INTERFACE IReadOnlyListOfBytes EXTENDS IPointerCollection

METHOD Find : BOOL
VAR_INPUT
	value : BYTE;
END_VAR
VAR_OUTPUT
	index : DINT;
END_VAR
END_METHOD

METHOD Get : BYTE
VAR_INPUT
	index : DINT;
END_VAR
END_METHOD

END_INTERFACE

(* stored: Version 1.1.0.1
   Itf IReadOnlyListOfBytes: Id {a843c369-9e00-00a1-32fa-d03c5ab85265}
   Method Find: Id {3f29ee40-326e-4872-b375-7e35c81e45f0}
   Method Get: Id {27925820-f345-0e43-1a3c-84ba47105d29} *)
